TEXTLIST TextListSpitUnitErrorid
  0 = 'no_error'
  1 = 'not_connected'
  2 = 'invalid_state'
  3 = 'homing_error'
  4 = 'trigger_limit'
  5 = 'io_error'
  6 = 'unknown_error'
  666 = 'emergency_error'
  7 = 'Drive_not_ready_for_operation'
   = ''
END_TEXTLIST

(* stored: Version 1.1.0.1, ProductVersion 3.1.4024.11
   TextList TextListSpitUnitErrorid: Id {81105d00-6345-44b9-9f8b-a5af46e38357} *)
